Staubli VAL3: getFbkPos.pgx

public program getFbkPos()
  local num l_i
begin
  for l_i=0 to nAxesSum-1
      //nScaleFact:电机转一圈角度（旋转轴）或前进距离（直线轴（mm））
      nDrvFbkPos[l_i]=nScaleFact[l_i]*aioGet(aiPosFbk[l_i])/nResolution[l_i]*nGearratio[l_i]
      nAxesPosFbk[l_i]=nDrvFbkPos[l_i]/nGearratio[l_i]
  endFor
end
